FUNCTION TryConvert_USINT_TO_DINT : BOOL
VAR_INPUT
	in : USINT;
	out : REFERENCE TO DINT;
END_VAR

out := USINT_TO_DINT(in);
TryConvert_USINT_TO_DINT := TRUE;

END_FUNCTION

(* stored: Version 1.1.0.1, ProductVersion 3.1.4024.12
   POU TryConvert_USINT_TO_DINT: Id {4e3cce6f-03c5-474e-9f46-b0ae139c6224}, SpecialFunc None *)
